FUNCTION_BLOCK FB_TransportA
VAR_INPUT
	bStop1 : BOOL;
	bStop2 : BOOL;
	bStop3 : BOOL;
END_VAR
VAR_OUTPUT
	bStopper1 : BOOL;
	bStopper2 : BOOL;
	bStopper3 : BOOL;
END_VAR
VAR
END_VAR

bStopper1 := bStop1;
bStopper2 := bStop2;
bStopper3 := bStop3;

END_FUNCTION_BLOCK

(* stored: Version 1.1.0.1, ProductVersion 3.1.4024.15
   POU FB_TransportA: Id {2057bef0-c93b-4182-bafe-9c938a2a7a84}, SpecialFunc None *)
